FUNCTION AGILOG_INFO : BOOL
VAR_INPUT
	// could be any data type, for array, only lreal is supported
	i_logData : ANY;
	// if to print time
	i_printTime :BOOL :=TRUE;
	//add a byte at the line end. 0: nothing, 1: new line, 2: space
	i_lineBreak :INT :=0;

END_VAR
VAR
	tmpData : LogDataType;
	checkIdx:INT;
END_VAR

IF NOT(GVL_RunTimeLogger.g_infoLogReady) THEN
	RETURN;
END_IF

// data decode
tmpData.m_dataType := i_logData.TypeClass;
tmpData.m_dataSize := MIN(i_logData.diSize,96);
tmpData.m_lineBreak := i_lineBreak;
tmpData.m_printTime := i_printTime;
tmpData.m_timeStamp := GVL_RunTimeLogger.g_localSystemTime.systemTime;
MEMCPY(ADR(tmpData.m_data), i_logData.pValue, tmpData.m_dataSize);

//add to buffer
FOR checkIdx :=1 TO 20 DO 
	IF TestAndSet(GVL_RunTimeLogger.g_infoLogBufferLock) THEN
		GVL_RunTimeLogger.g_infoLogBuffer[GVL_RunTimeLogger.g_infoLogBufferInPtr] := tmpData;
		// step pointer
		IF GVL_RunTimeLogger.g_infoLogBufferInPtr >= GVL_RunTimeLogger.g_infoLogBufferSize THEN
			GVL_RunTimeLogger.g_infoLogBufferInPtr := 1;
		ELSE
			GVL_RunTimeLogger.g_infoLogBufferInPtr:=GVL_RunTimeLogger.g_infoLogBufferInPtr+1;
		END_IF
		GVL_RunTimeLogger.g_infoLogBufferLock := false;
		EXIT;
	END_IF
END_FOR

END_FUNCTION

(* stored: Version 1.1.0.1, ProductVersion 3.1.4024.12
   POU AGILOG_INFO: Id {d769d76e-905c-45d8-8351-63f42bd44cee}, SpecialFunc None *)
